(*!
<summary>Classifies diagnostic records for filtering, numbering and output severity.</summary>
<description>
Categories increase from DEBUG to CRITICAL_ERROR. Mapping to a physical logging service is backend-specific;
category alone does not change PLC execution.
</description>
*)
(*
SPDX-FileCopyrightText: © 2026 Oleksandr Tiutyk <trofimich@gmail.com>
SPDX-License-Identifier: MIT
License: https://opensource.org/license/mit
*)

{attribute 'qualified_only'}
{attribute 'strict'}
{attribute 'to_string'}
TYPE LOG_CATEGORY :
(
	DEBUG := 0,
	INFORMATION,
	WARNING,
	ERROR,
	CRITICAL_ERROR
);
END_TYPE

(* stored: Version 1.1.0.1
   DUT LOG_CATEGORY: Id {9661d15e-b34f-4e09-a7e5-cf9e937438a5} *)
